// TIA Portal V19 export
TYPE "Positioning_EPOS_Machine_Wng"
// stored: Access Published
   STRUCT
      NotAutReady : Bool;   // Machine is NOT ready for automatic start
      Minus_CndMissing : Bool;   // Lack of conditions for movement in negative direction
      Plus_CndMissing : Bool;   // Lack of conditions for movement in positive direction
      S120_Warning : Bool;   // SINAMICS S120 warning presence
      Ax_NotHomed : Bool;   // Axis is not homed / referenced
      Ax_FlyingHome : Bool;   // Flying homing could not be started
      Ax_SwLimitMinus : Bool;   // Negative software limit reached / exceeded
      Ax_SwLimitPlus : Bool;   // Positive software limit reached / exceeded
   END_STRUCT;
END_TYPE
